// TwinCAT 3 PLC project plc1
// ProgramVersion: 3.1.4024.0
// libraries:
//   Tc2_Standard, * (Beckhoff Automation GmbH)
//   Tc2_System, * (Beckhoff Automation GmbH)
//   Tc3_Module, * (Beckhoff Automation GmbH)
// project tree:
//   GVL/ GVL.TcGVL
//   / PlcTask.TcTTO
//   POUs/ FbdRule.TcPOU, MAIN.TcPOU, Pine_Branch_Test.TcPOU, StDrool.TcPOU
// real-time tasks:
//   TASK PlcTask: cycle T#10ms, priority 20, ADS port 350

CONFIGURATION plc1
    RESOURCE PLC ON TwinCAT3
        TASK PlcTask(INTERVAL := T#10ms, PRIORITY := 20);
        PROGRAM MAIN WITH PlcTask : MAIN;
    END_RESOURCE
END_CONFIGURATION

// ---- GVL/GVL.TcGVL
{attribute 'qualified_only'}
VAR_GLOBAL
	
	CoolGuyAlert : BOOL;
	DiskGolfMaster : BOOL;
	
END_VAR

// ---- POUs/MAIN.TcPOU
PROGRAM MAIN
VAR
	bing: BOOL;
	bong: BOOL;
	ProfessorOak: INT;
	givespokemon: INT;
END_VAR

bing := bong;



ProfessorOak := givespokemon;

END_PROGRAM

// ---- POUs/FbdRule.TcPOU
PROGRAM FbdRule
VAR
	alex: BOOL;
	coffee: BOOL;
	workGetsDone: BOOL;
END_VAR

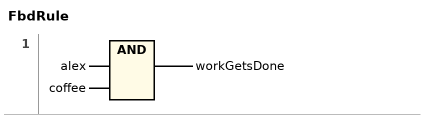
// NETWORK 1
workGetsDone := alex AND coffee;

END_PROGRAM

// ---- POUs/Pine_Branch_Test.TcPOU
PROGRAM Pine_Branch_Test
VAR
END_VAR

// Pine branch test by Alan from his laptop.

END_PROGRAM

// ---- POUs/StDrool.TcPOU
PROGRAM StDrool
VAR
	CaseCool: INT;
	YellowMinions: INT;
	WorkAtUS: INT;
	JustinAndAlex: INT;
	lookFly: INT;
END_VAR

CASE CaseCool OF 
	0:
		YellowMinions := WorkAtUS;
		
	1: 
		//free cars for everybody
		
	2: 
		JustinAndAlex := lookFly;
		
		
END_CASE

END_PROGRAM
